SYSTEM TEST_FIFO (* Test FIFO_UINT in a RMT_DEV *)
  (* Standard: 61499-1 *)
  (* Version 0.0, 2005-12-13, JHC, Holobloc Inc *)
  DEVICE GUI : FRAME_DEVICE(BOUNDS := [100,100,200,150], GRID := [1,2])
    RESOURCE INPUT : PANEL_RESOURCE
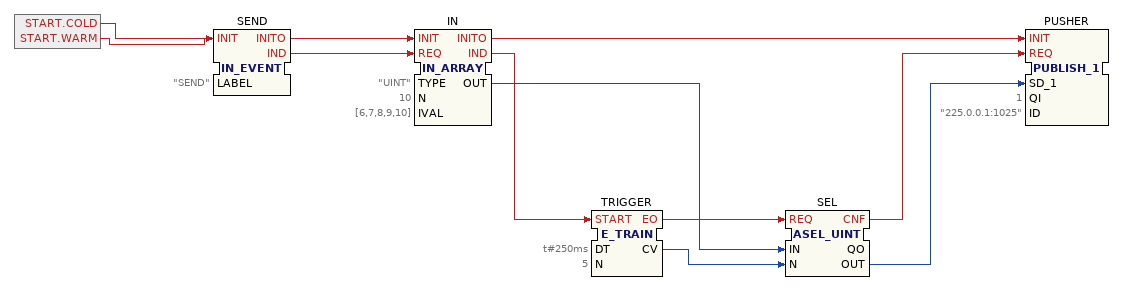
      FBS
        SEND : IN_EVENT(LABEL := "SEND");
        IN : IN_ARRAY(TYPE := "UINT", N := 10, IVAL := [6,7,8,9,10]);
        PUSHER : PUBLISH_1(QI := 1, ID := "225.0.0.1:1025");
        TRIGGER : E_TRAIN(DT := t#250ms, N := 5);
        SEL : ASEL_UINT;
      END_FBS
      EVENT_CONNECTIONS
        START.COLD TO SEND.INIT;
        START.WARM TO SEND.INIT;
        SEND.INITO TO IN.INIT;
        SEND.IND TO IN.REQ;
        IN.INITO TO PUSHER.INIT;
        IN.IND TO TRIGGER.START;
        TRIGGER.EO TO SEL.REQ;
        SEL.CNF TO PUSHER.REQ;
      END_CONNECTIONS
      DATA_CONNECTIONS
        IN.OUT TO SEL.IN;
        TRIGGER.CV TO SEL.N;
        SEL.OUT TO PUSHER.SD_1;
      END_CONNECTIONS
    END_RESOURCE
    RESOURCE OUTPUT : PANEL_RESOURCE
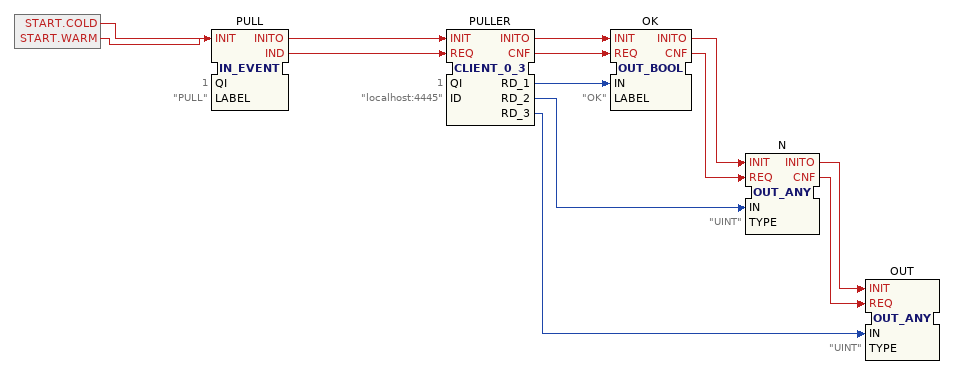
      FBS
        PULLER : CLIENT_0_3(QI := 1, ID := "localhost:4445");
        PULL : IN_EVENT(QI := 1, LABEL := "PULL");
        OK : OUT_BOOL(LABEL := "OK");
        N : OUT_ANY(TYPE := "UINT");
        OUT : OUT_ANY(TYPE := "UINT");
      END_FBS
      EVENT_CONNECTIONS
        START.COLD TO PULL.INIT;
        START.WARM TO PULL.INIT;
        PULL.INITO TO PULLER.INIT;
        PULL.IND TO PULLER.REQ;
        PULLER.INITO TO OK.INIT;
        PULLER.CNF TO OK.REQ;
        OK.INITO TO N.INIT;
        OK.CNF TO N.REQ;
        N.INITO TO OUT.INIT;
        N.CNF TO OUT.REQ;
      END_CONNECTIONS
      DATA_CONNECTIONS
        PULLER.RD_1 TO OK.IN;
        PULLER.RD_2 TO N.IN;
        PULLER.RD_3 TO OUT.IN;
      END_CONNECTIONS
    END_RESOURCE
  END_DEVICE
  DEVICE REMOTE : RMT_DEV
    RESOURCE FIFO_RES : EMB_RES
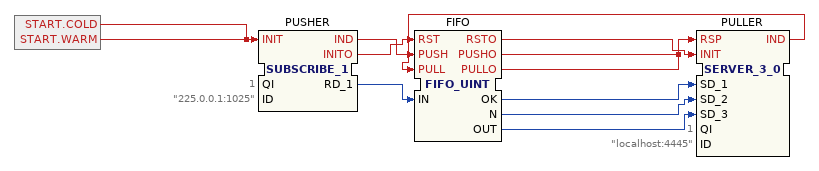
      FBS
        FIFO : FIFO_UINT;
        PUSHER : SUBSCRIBE_1(QI := 1, ID := "225.0.0.1:1025");
        PULLER : SERVER_3_0(QI := 1, ID := "localhost:4445");
      END_FBS
      EVENT_CONNECTIONS
        START.COLD TO PUSHER.INIT;
        START.WARM TO PUSHER.INIT;
        FIFO.PULLO TO PULLER.RSP;
        PULLER.IND TO FIFO.PULL;
        PUSHER.IND TO FIFO.PUSH;
        FIFO.PUSHO TO PULLER.RSP;
        PUSHER.INITO TO FIFO.RST;
        FIFO.RSTO TO PULLER.INIT;
      END_CONNECTIONS
      DATA_CONNECTIONS
        PUSHER.RD_1 TO FIFO.IN;
        FIFO.OK TO PULLER.SD_1;
        FIFO.N TO PULLER.SD_2;
        FIFO.OUT TO PULLER.SD_3;
      END_CONNECTIONS
    END_RESOURCE
  END_DEVICE
END_SYSTEM
